KUKA KRL program: RUNFILE.src, RUNFILE.dat

--- RUNFILE.src ---
&ACCESS RVP
&REL 102
&PARAM TEMPLATE = C:\KRC\Roboter\Template\vorgabe
&PARAM EDITMASK = *
DEF RUNFILE( )

DECL BOOL RESPONSE
DECL INT HANDLE
DECL STATE_T SC_T
DECL INT J

;FOLD INI
  ;FOLD BASISTECH INI
    GLOBAL INTERRUPT DECL 3 WHEN $STOPMESS==TRUE DO IR_STOPM ( )
    INTERRUPT ON 3
    BAS (#INITMOV,0 )
  ;ENDFOLD (BASISTECH INI)
  ;FOLD USER INI
    ;Make your modifications here
  ;ENDFOLD (USER INI)
;ENDFOLD (INI)


;$BASE=BASE_DATA[1]
;$TOOL=TOOL_DATA[7]


;FOR J=1 TO 6
;  $ACC_AXIS[J]=25
;  $VEL_AXIS[J]=25
;ENDFOR

;$STIFFNESS.strategy = 10
;$STIFFNESS.commit = TRUE


RESPONSE = STARTIMPEDANCE(FALSE)

PTP $POS_ACT_MES


TCP_CONNECTED = FALSE
FCACTIVE = FALSE    ; force a reset of force control

;CCLOSE(HANDLE,SC_T)
IF USE_SERIAL THEN
  ; Open serial connection
  COPEN(:SER_3, HANDLE)
  IF HANDLE==0 THEN
    HALT
  ENDIF
ELSE
  ; receive structure
  CRPI_REC_TEXT[1].s[] = "CRPICommand.CRPIData.CMD"
  CRPI_REC_TEXT[2].s[] = "CRPICommand.CRPIData.Values.V1"
  CRPI_REC_TEXT[3].s[] = "CRPICommand.CRPIData.Values.V2"
  CRPI_REC_TEXT[4].s[] = "CRPICommand.CRPIData.Values.V3"
  CRPI_REC_TEXT[5].s[] = "CRPICommand.CRPIData.Values.V4"
  CRPI_REC_TEXT[6].s[] = "CRPICommand.CRPIData.Values.V5"
  CRPI_REC_TEXT[7].s[] = "CRPICommand.CRPIData.Values.V6"
  CRPI_REC_TEXT[8].s[] = "CRPICommand.CRPIData.Values.V7"
  CRPI_REC_TEXT[9].s[] = "CRPICommand.CRPIData.Values.V8"
  CRPI_REC_TEXT[10].s[] = "CRPICommand.CRPIData.Values.V9"
  CRPI_REC_TEXT[11].s[] = "CRPICommand.CRPIData.Values.V10"
  CRPI_REC_TEXT[12].s[] = "CRPICommand.CRPIData"
  CRPI_SENSOR_NAME[]="CRPICommand"

  ; Open Ethernet connection
  IF NOT USE_SERIAL THEN
    WHILE NOT TCP_CONNECTED
      errint = EKX_open(CRPI_SENSOR_NAME[])
      ;EKX_handleerror(errint)
      IF errint == eioc_error THEN
        ; USED TO BE HALT
      ELSE
        TCP_CONNECTED = TRUE
      ENDIF
    ENDWHILE
  ENDIF

;  errint = EKX_open(CRPI_SENSOR_NAME[])
;  EKX_handleerror(errint)
;  IF errint == eioc_error THEN
;    HALT
;  ELSE
;    TCP_CONNECTED = TRUE
;  ENDIF

  HANDLE = 0
ENDIF

LOOP
  RESPONSE = LISTEN( HANDLE )

  IF NOT USE_SERIAL THEN
    WHILE NOT TCP_CONNECTED
      errint = EKX_open(CRPI_SENSOR_NAME[])
      ;EKX_handleerror(errint)
      IF errint == eioc_error THEN
        ; USED TO BE HALT
      ELSE
        TCP_CONNECTED = TRUE
      ENDIF
    ENDWHILE
  ENDIF

ENDLOOP

IF USE_SERIAL THEN
  ; Close serial connection
  CCLOSE( HANDLE, SC_T )
ELSE
  ; Close Ethernet connection
  errbl = EKX_close(CRPI_SENSOR_NAME[])
  IF errbl == FALSE THEN
    HALT
  ENDIF
ENDIF

IF SC_T.RET1<>#CMD_OK THEN
  HALT
ENDIF

;FOLD PTP HOME  Vel= 100 % DEFAULT;%{PE}%MKUKATPBASIS,%CMOVE,%VPTP,%P 1:PTP, 2:HOME, 3:, 5:100, 7:DEFAULT
$BWDSTART = FALSE
PDAT_ACT=PDEFAULT
FDAT_ACT=FHOME
BAS (#PTP_PARAMS,100 )
$H_POS=XHOME
PTP  XHOME
;ENDFOLD

END

--- RUNFILE.dat ---
&ACCESS RVP
&REL 102
&PARAM TEMPLATE = C:\KRC\Roboter\Template\vorgabe
&PARAM EDITMASK = *
DEFDAT  RUNFILE
;FOLD EXTERNAL DECLARATIONS;%{PE}%MKUKATPBASIS,%CEXT,%VCOMMON,%P
;FOLD BASISTECH EXT;%{PE}%MKUKATPBASIS,%CEXT,%VEXT,%P
EXT  BAS (BAS_COMMAND  :IN,REAL  :IN )
DECL INT SUCCESS
;ENDFOLD (BASISTECH EXT)
;FOLD USER EXT;%{E}%MKUKATPUSER,%CEXT,%VEXT,%P
;Make here your modifications

;ENDFOLD (USER EXT)
;ENDFOLD (EXTERNAL DECLARATIONS)
DECL BASIS_SUGG_T LAST_BASIS={POINT1[] "P5                      ",POINT2[] "P5                      ",CP_PARAMS[] "CPDAT0                  ",PTP_PARAMS[] "PDAT5                   ",CONT[] "                        ",CP_VEL[] "2.0                     ",PTP_VEL[] "25                      ",SYNC_PARAMS[] "SYNCDAT                 ",SPL_NAME[] "S0                      "}
DECL E6POS XP1={X 0.0639737174,Y -687.130188,Z 128.787796,A 89.9691772,B -0.287573099,C -179.996002,S 6,T 25,E1 -0.000798225403,E2 0.0,E3 0.0,E4 0.0,E5 0.0,E6 0.0}
DECL FDAT FP1={TOOL_NO 7,BASE_NO 0,IPO_FRAME #BASE,POINT2[] " ",TQ_STATE FALSE}
DECL PDAT PPDAT1={VEL 100.0,ACC 100.0,APO_DIST 100.0,APO_MODE #CPTP}
DECL E6POS XP2={X 554.680115,Y -367.072601,Z 395.465302,A 0.00234176009,B 0.000156519294,C 44.9950409,S 2,T 0,E1 -89.9905167,E2 0.0,E3 0.0,E4 0.0,E5 0.0,E6 0.0}
DECL FDAT FP2={TOOL_NO 1,BASE_NO 0,IPO_FRAME #BASE,POINT2[] " ",TQ_STATE FALSE}
DECL PDAT PPDAT2={VEL 100.0,ACC 100.0,APO_DIST 100.0,APO_MODE #CPTP}
DECL E6POS XP3={X 554.693481,Y -200.003296,Z 395.334015,A 0.0104174297,B 0.00705960579,C 45.0026398,S 2,T 0,E1 -89.9838562,E2 0.0,E3 0.0,E4 0.0,E5 0.0,E6 0.0}
DECL FDAT FP3={TOOL_NO 1,BASE_NO 0,IPO_FRAME #BASE,POINT2[] " ",TQ_STATE FALSE}
DECL PDAT PPDAT3={VEL 100.0,ACC 100.0,APO_DIST 100.0,APO_MODE #CPTP}
DECL E6POS XP4={X 554.701721,Y -50.0167694,Z 395.272308,A 0.00931109954,B 0.0131273204,C 45.0018997,S 2,T 0,E1 -89.980217,E2 0.0,E3 0.0,E4 0.0,E5 0.0,E6 0.0}
DECL FDAT FP4={TOOL_NO 1,BASE_NO 0,IPO_FRAME #BASE,POINT2[] " ",TQ_STATE FALSE}
DECL PDAT PPDAT4={VEL 100.0,ACC 100.0,APO_DIST 100.0,APO_MODE #CPTP}
DECL E6POS XP5={X 554.723022,Y -0.00272168103,Z 395.199402,A 0.0169154797,B 0.0238184407,C 45.0061798,S 2,T 0,E1 -89.9762497,E2 0.0,E3 0.0,E4 0.0,E5 0.0,E6 0.0}
DECL FDAT FP5={TOOL_NO 1,BASE_NO 0,IPO_FRAME #BASE,POINT2[] " ",TQ_STATE FALSE}
DECL PDAT PPDAT5={VEL 100.0,ACC 100.0,APO_DIST 100.0,APO_MODE #CPTP}

ENDDAT
